TYPE ST_MyStruct :
STRUCT
	iVal1	: INT;
	iVal2	: INT;
	iVal3	: INT;
END_STRUCT
END_TYPE

(* stored: Version 1.1.0.1, ProductVersion 3.1.4024.12
   DUT ST_MyStruct: Id {f93a59ff-e066-4f74-afc4-a8680a6d6d59} *)
